Universal Robots PolyScope program: Bag_mixing_v5.urp

Program Bag_mixing_v5 (installation=default directory=/programs/usbdisk/analysing-mixing-of-single-use-bags createdIn=5.5.0 lastSavedIn=5.16.0 robotSerialNumber=20225205248)
Calibrated DH parameters: a=[0.00004, -0.603342, -0.567862, 0.000011, -0.000063, 0]; d=[0.180788, 1523.697461, -1534.664592, 11.140954, 0.119775, 0.115531]; alpha=[1.570213, 0.000068, 0.005575, 1.569427, -1.569944, 0]; deltaTheta=[-0.000001, 0.169538, 6.006402, 0.107243, 0, -0.000001]
InitVariablesNode
BeforeStart
  Timer (action=Stop) variable(name=timer_1)
  URCap F/T Sensor Command (ATI Axia Force/Torque Sensor, ATI Industrial Automation) dataModel(running=Enable)
  URCap F/T Sensor Options (ATI Axia Force/Torque Sensor, ATI Industrial Automation) dataModel(RADIO_SELECTED=true, NETFT_STATUS=00000000, RDT_RATE=500, AXIA_STATUS=00000000, LOGGING_LEVEL=2, AXIA_SELECTED=true, AXIA_FILTER_IDX=1)
  frequency := 0
  gap_width := 0
  stroke := 0
  duration := 0
  var_4 := 0
  thrd_1 := 0
  thrd_2 := 0
  p_amp := 0
  p_minreached := False
Robot Program (runOnlyOnce=false)
  URCap Find Visual Offset (Robotiq_Wrist_Camera, Robotiq Inc.) dataModel(tagModel=[{"_featureName":"bag_mix_plane","_automaticMoveEnabled":true,"_ignoreSnapshotPositionEnabled":false,"_skipCloseSnapshotPositionEnabled":false}]); state(isChildrenLocked=true)
    URCap If tag found (Robotiq_Wrist_Camera, Robotiq Inc.)
      URCap Apply Visual Offset (Robotiq_Wrist_Camera, Robotiq Inc.)
        'Insert actions here'
    URCap If tag not found (Robotiq_Wrist_Camera, Robotiq Inc.)
      Placeholder
    URCap If tag found (Robotiq_Wrist_Camera, Robotiq Inc.)
      URCap Apply Visual Offset (Robotiq_Wrist_Camera, Robotiq Inc.) dataModel(tagModel=[{"_featureName":"bag_mix_plane","_appliedEverywhere":false}])
        err_rx := bag_mix_plane[3] - 1 * 3.14159/180
        Wait Sleep waitTime=0.5
        Wait Sleep waitTime=0.5
        bag_mix_plane := p[bag_mix_plane[0], bag_mix_plane[1], bag_mix_plane[2], 0, 0, bag_mix_plane[5]]
        plane_rot := rotvec2rpy([err_rx, 0, bag_mix_plane[5]])
        rx_d := 180 - r2d(plane_rot[0])
        popup_msg := str_cat("Ready to receive mixing values. Angle about X: ", rx_d)
        Popup Message (haltProgram=false inputType=Variable) variable=popup_msg
        Loop Forever
          p_minreached := False
          Wait Sleep waitTime=0.5
          var_1 := socket_open("192.168.0.32", 30000)
          Loop While (checkContinuously=false) expression=var_1 ≟  False
            var_1 := socket_open("192.168.0.32", 30000)
            Wait Sleep waitTime=0.5
          Script: socket_send_string("send_program_parameters")
          var_2 := socket_read_ascii_float(5)
          Script: socket_close()
          var_1 := False
          If var_2[0] ≠ 0
            frequency := var_2[1]
            gap_width := var_2[2]
            stroke := var_2[3]
            duration := var_2[4]
            angle_user_inp := var_2[5]
          If (rx_d < 360) and (rx_d > 358)
            rx_d := 0
          rx_d_lim_down := rx_d - 2
          rx_d_lim_up := rx_d + 2
          If (angle_user_inp < rx_d_lim_down) or (angle_user_inp >rx_d_lim_up)
            Popup Error (haltProgram=false message=Angle of the plane doesn't match the user input! inputType=Text)
            Halt
          If (gap_width < 2) or (gap_width > 50)
            Popup Error (haltProgram=true message=Wrong value for gap width! inputType=Text)
          gap_width := gap_width*0.001
          If (frequency ≤ 0) or (frequency > 7)
            Popup Error (haltProgram=true message=Wrong value for the frequency! inputType=Text)
          stroke := stroke*0.001
          If (stroke ≤ 0) or (stroke > 25)
            Popup Error (haltProgram=true message=Wrong value for the lifting height! inputType=Text)
          p_amp := stroke/2
          If (angle_user_inp < 0) or (angle_user_inp > 50)
            Popup Error (haltProgram=true message=Wrong value for the angle of mixing plane! inputType=Text)
          mixer := p[mixer[0], mixer[1], mixer[2], 3.14159 - angle_user_inp * 3.14159/180 - 0.0, mixer[4] - 0.03, mixer[5] - 0.008]
          p_min0 := p[-0.020, -0.055, - gap_width - stroke, 0, -0, 0]
          p_max_safe := p[p_min0[0], p_min0[1], -0.2, p_min0[3], p_min0[4], p_min0[5]]
          If p_minreached≟ False
            MoveJ speed 60 deg/s, acceleration 80 deg/s^2 (useActiveTCP=true) feature=mixer
              Waypoint Variable (Variable): variable(name=p_max_safe)
              Waypoint Variable (Variable): variable(name=p_min0)
            Popup Warning (haltProgram=false message=Initial position reached. Start movement? inputType=Text)
            p_minreached := True
          var_3 := socket_open("192.168.0.32", 30001)
          Loop While (checkContinuously=false) expression=var_3 ≟ False
            Wait Sleep waitTime=0.2
            var_3 := socket_open("192.168.0.32", 30001)
          Script: socket_send_string("motion_started")
          Script: socket_close()
          URCap F/T Sensor Command (ATI Axia Force/Torque Sensor, ATI Industrial Automation) dataModel(running=Bias)
          Loop While (checkContinuously=false) expression=timer_1 < duration
            MoveL speed 8 mm/s, acceleration 1200 mm/s^2 (useActiveTCP=true) feature=mixer
              Waypoint Variable (Variable): variable=p_min0
              Script: sync()
              Waypoint Variable (Variable): variable=p_min0
            Wait Sleep waitTime=0.01
          p_minreached := False
          Wait Sleep waitTime=3
          MoveJ speed 60 deg/s, acceleration 80 deg/s^2 (useActiveTCP=true) feature=Base
            Waypoint Waypoint_1: TCP in base x=-30.82 y=-630.657 z=294.621 mm, rx=3.1416 ry=0 rz=0 rad; joints [71.228, -94.449, 114.942, -110.446, -89.723, 161.382] deg; TCP offset x=0 y=0 z=180 mm, rx=0 ry=0 rz=0 rad
    URCap If tag not found (Robotiq_Wrist_Camera, Robotiq Inc.)
      Popup Message (haltProgram=false message=Tag not found! inputType=Text)
Thread Thread_2 (runOnlyOnce=false)
  Wait Sleep waitTime=2
  timer_1 := 0
  t := 0
  pi := 3.14159
  alpha := 0.5
  If p_minreached≟ True
    Timer (action=Start) variable=timer_1
    t_now := 0
    t_start := get_steptime()
    Script: path_offset_enable()
    Script: path_offset_set_alpha_filter(alpha)
    Loop While (checkContinuously=false) expression=timer_1 < duration
      p1 := p_amp*(1-cos(2*pi*frequency*t))
      t_now := 0
      t := t+ 0.002
      Script: path_offset_set([0,0,p1,0,0,0], 2)
      Script: sync()
SuppressedNode
  SubProgram calculating_new_mix_plane (keepSynchronizedWithDisk=false) programFile=/programs/Bag_mixing/calculating_new_mix_plane.urp
    URCap Find Visual Offset (Robotiq_Wrist_Camera, Robotiq Inc.) dataModel(tagModel=[{"_featureName":"bag_mix_plane","_automaticMoveEnabled":true,"_ignoreSnapshotPositionEnabled":false,"_skipCloseSnapshotPositionEnabled":false}]); state(isChildrenLocked=true)
      URCap If tag found (Robotiq_Wrist_Camera, Robotiq Inc.)
        URCap Apply Visual Offset (Robotiq_Wrist_Camera, Robotiq Inc.)
          'Insert actions here'
      URCap If tag not found (Robotiq_Wrist_Camera, Robotiq Inc.)
        Placeholder
      URCap If tag found (Robotiq_Wrist_Camera, Robotiq Inc.)
        URCap Apply Visual Offset (Robotiq_Wrist_Camera, Robotiq Inc.) dataModel(tagModel=[{"_featureName":"bag_mix_plane","_appliedEverywhere":false}])
          err_rx := bag_mix_plane[3] - 2 * 3.14159/180
          err_ry := bag_mix_plane[4] + 0.8 * 3.14159/180
          bag_mix_plane := p[bag_mix_plane[0], bag_mix_plane[1], bag_mix_plane[2], err_rx, err_ry, bag_mix_plane[5]]
          plane_rot := rotvec2rpy([err_rx, err_ry, bag_mix_plane[5]])
          rx_d := 180 - r2d(plane_rot[0])
          popup_msg := str_cat("Angle about X: ", rx_d)
          Popup Message (haltProgram=false inputType=Variable) variable=popup_msg
      URCap If tag not found (Robotiq_Wrist_Camera, Robotiq Inc.)
        Popup Message (haltProgram=false message=Tag not found! inputType=Text)
